# B&R Automation Studio project SampleProject
Automation Studio 

## Configuration Config1

### Cpu.per - X20CP3173/Cpu.per
```
TaskConfiguration:
  Task CyclicTask (TaskClass=cyclic, CycleTime=10ms, Priority=1)
    Property (Source=MainProgram/Main.st)
  Task InitTask (TaskClass=init, Priority=0)
    Property (Source=MainProgram/Main.st)
```

## Logical view

### GlobalTypes.typ
```iecst
TYPE
	MotorStateEnum : (
		MOTORSTATE_IDLE,
		MOTORSTATE_STARTING,
		MOTORSTATE_RUNNING,
		MOTORSTATE_STOPPING,
		MOTORSTATE_FAULT
	);
	MotorConfigType : STRUCT
		MaxSpeed    : REAL := 3000.0;  (* Maximum motor speed [rpm] *)
		RampTime    : TIME := T#2s;    (* Acceleration ramp time *)
		FaultLimit  : REAL := 3500.0;  (* Overspeed fault threshold [rpm] *)
	END_STRUCT;
END_TYPE
```

### GVL_Main.var
```iecst
VAR_GLOBAL
	(* GVL_Main *)
	gMotorSpeed : REAL := 0.0;  (* Actual motor speed [rpm] *)
	gFault      : BOOL;         (* System fault flag *)
	gCycleCount : DINT := 0;    (* Total cycle counter *)
END_VAR
```

### Program Logical/MainProgram (MainProgram, version 4)

#### Main.st - Main
```iecst
(*
 * MainProgram — Main cyclic program
 * Coordinates motor start/stop sequence using a state machine.
 *)

(* _INIT section *)
State := MOTORSTATE_IDLE;
gMotorSpeed := 0.0;
gFault := FALSE;

(* _CYCLIC section *)
CASE State OF

	MOTORSTATE_IDLE:
		gMotorSpeed := 0.0;
		IF StartCmd AND NOT gFault THEN
			State := MOTORSTATE_STARTING;
			TON_ramp.PT := Config.RampTime;
			TON_ramp.IN := TRUE;
			TON_ramp();
		END_IF

	MOTORSTATE_STARTING:
		TON_ramp.IN := TRUE;
		TON_ramp();
		gMotorSpeed := gMotorSpeed + 100.0;
		IF gMotorSpeed >= Config.MaxSpeed THEN
			gMotorSpeed := Config.MaxSpeed;
			State := MOTORSTATE_RUNNING;
		END_IF
		IF gMotorSpeed > Config.FaultLimit THEN
			gFault := TRUE;
			State := MOTORSTATE_FAULT;
		END_IF

	MOTORSTATE_RUNNING:
		IF StopCmd THEN
			State := MOTORSTATE_STOPPING;
			TON_ramp.IN := FALSE;
			TON_ramp();
		END_IF
		IF gMotorSpeed > Config.FaultLimit THEN
			gFault := TRUE;
			State := MOTORSTATE_FAULT;
		END_IF

	MOTORSTATE_STOPPING:
		gMotorSpeed := gMotorSpeed - 100.0;
		IF gMotorSpeed <= 0.0 THEN
			gMotorSpeed := 0.0;
			State := MOTORSTATE_IDLE;
		END_IF

	MOTORSTATE_FAULT:
		gMotorSpeed := 0.0;
		TON_ramp.IN := FALSE;
		TON_ramp();
		IF NOT gFault THEN
			State := MOTORSTATE_IDLE;
		END_IF

END_CASE

gCycleCount := gCycleCount + 1;
```

#### Local.var - Local
```iecst
VAR
	State       : MotorStateEnum;
	Config      : MotorConfigType;
	StartCmd    : BOOL;
	StopCmd     : BOOL;
	TON_ramp    : TON;
END_VAR
```

### Program Logical/MotorControl (MotorControl, version 4)

#### MotorControl.st - Main
```iecst
(*
 * MotorControl FB — Controls motor speed with ramp and fault detection
 *)
FUNCTION_BLOCK MotorControl

R_TRIG_start.CLK := Enable;
R_TRIG_start();

IF Enable THEN
	TON_delay.IN := TRUE;
	TON_delay.PT := T#500ms;
	TON_delay();
	IF TON_delay.Q THEN
		ActualSpeed := SpeedSetpoint;
		Running := TRUE;
	END_IF
ELSE
	TON_delay.IN := FALSE;
	TON_delay();
	ActualSpeed := 0.0;
	Running := FALSE;
END_IF

gMotorSpeed := ActualSpeed;

END_FUNCTION_BLOCK
```

#### MotorControl.var - Local
```iecst
VAR_INPUT
	Enable      : BOOL;
	SpeedSetpoint : REAL;   (* Speed setpoint [rpm] *)
END_VAR
VAR_OUTPUT
	ActualSpeed : REAL;     (* Measured speed [rpm] *)
	Running     : BOOL;
END_VAR
VAR
	TON_delay   : TON;
	R_TRIG_start : R_TRIG;
END_VAR
```
